# B&R Automation Studio project DuctLines (part 13)

#### Cyclic.ld
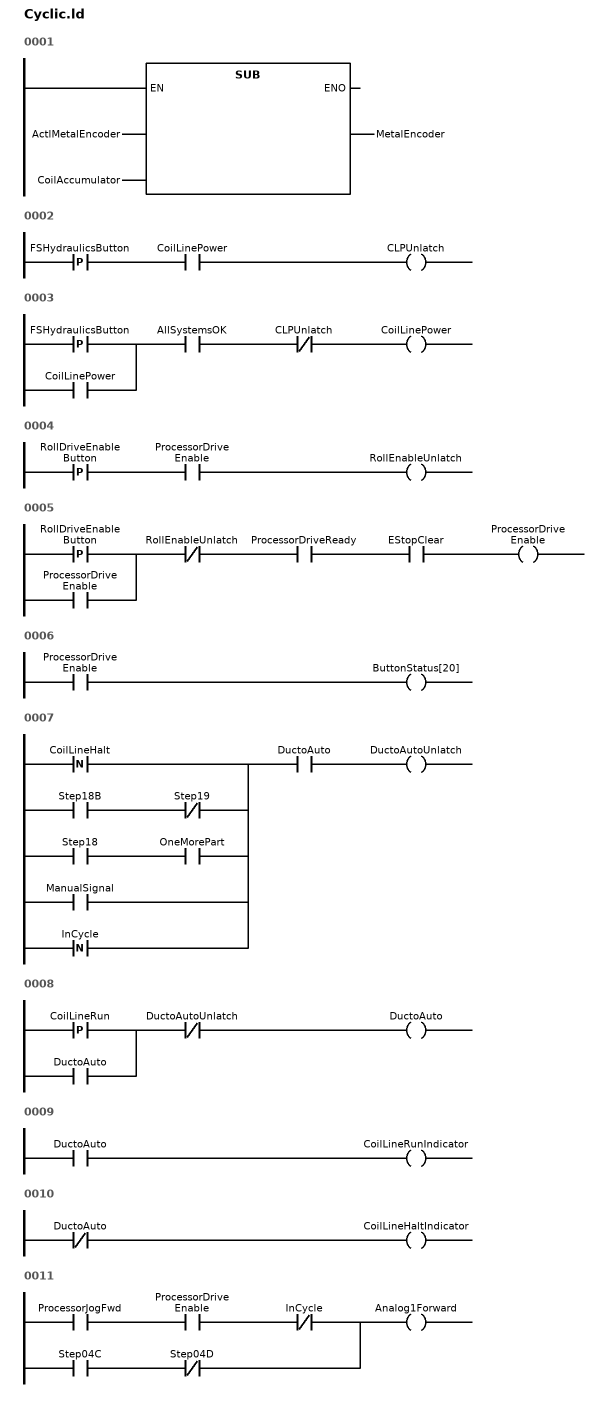
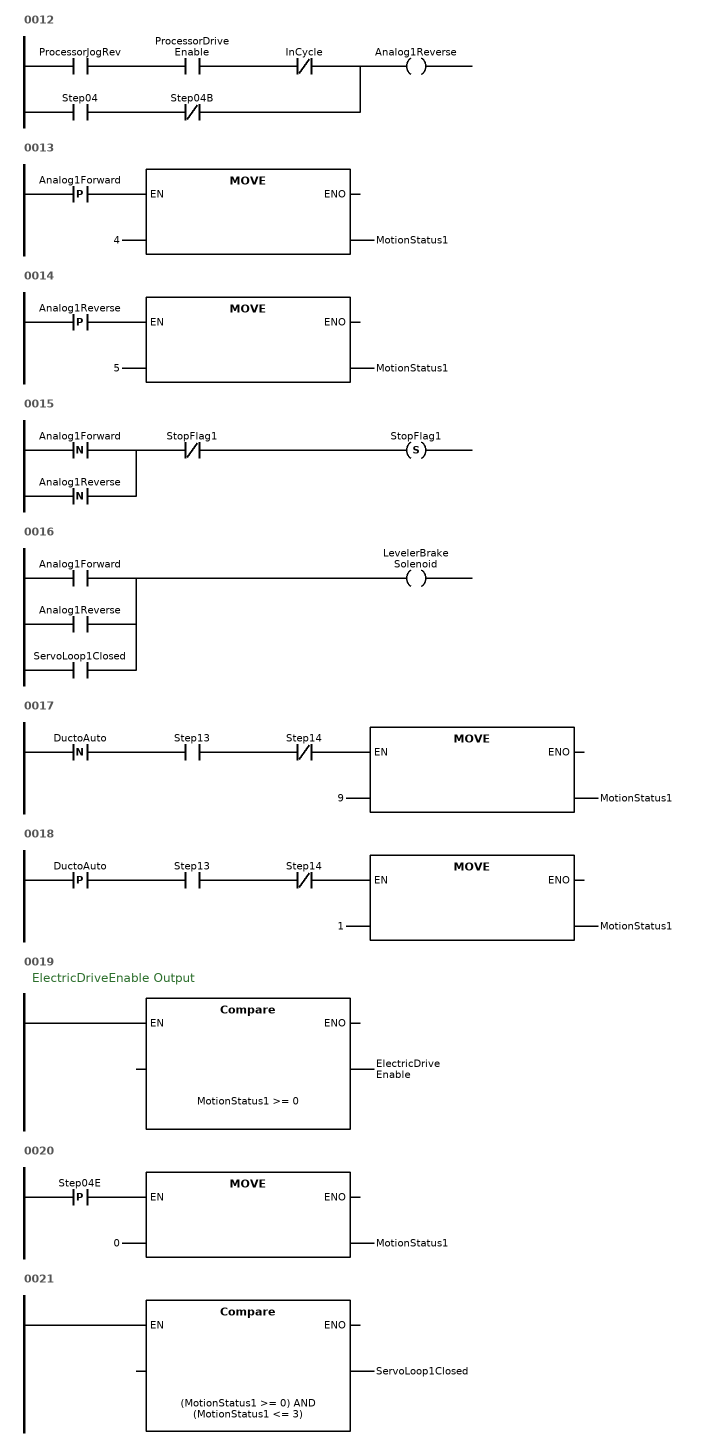
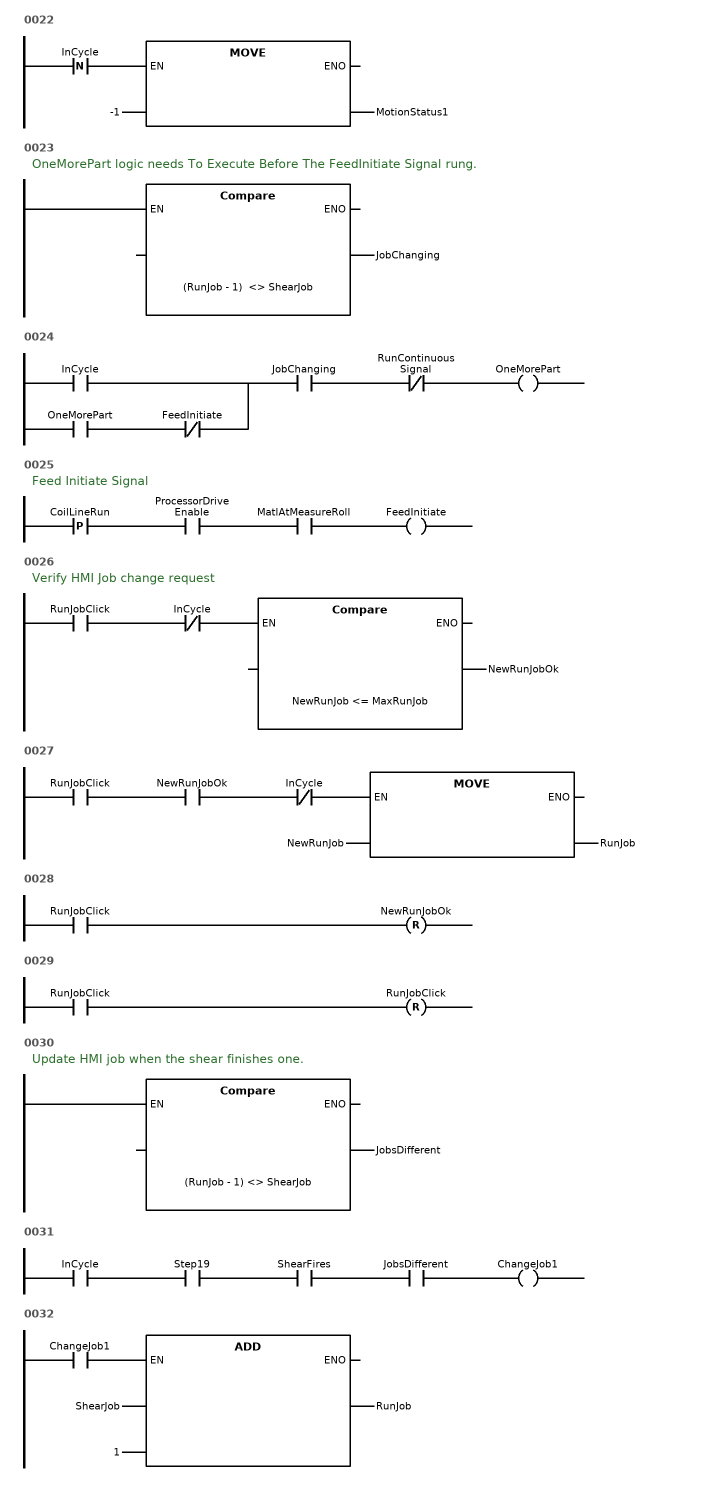
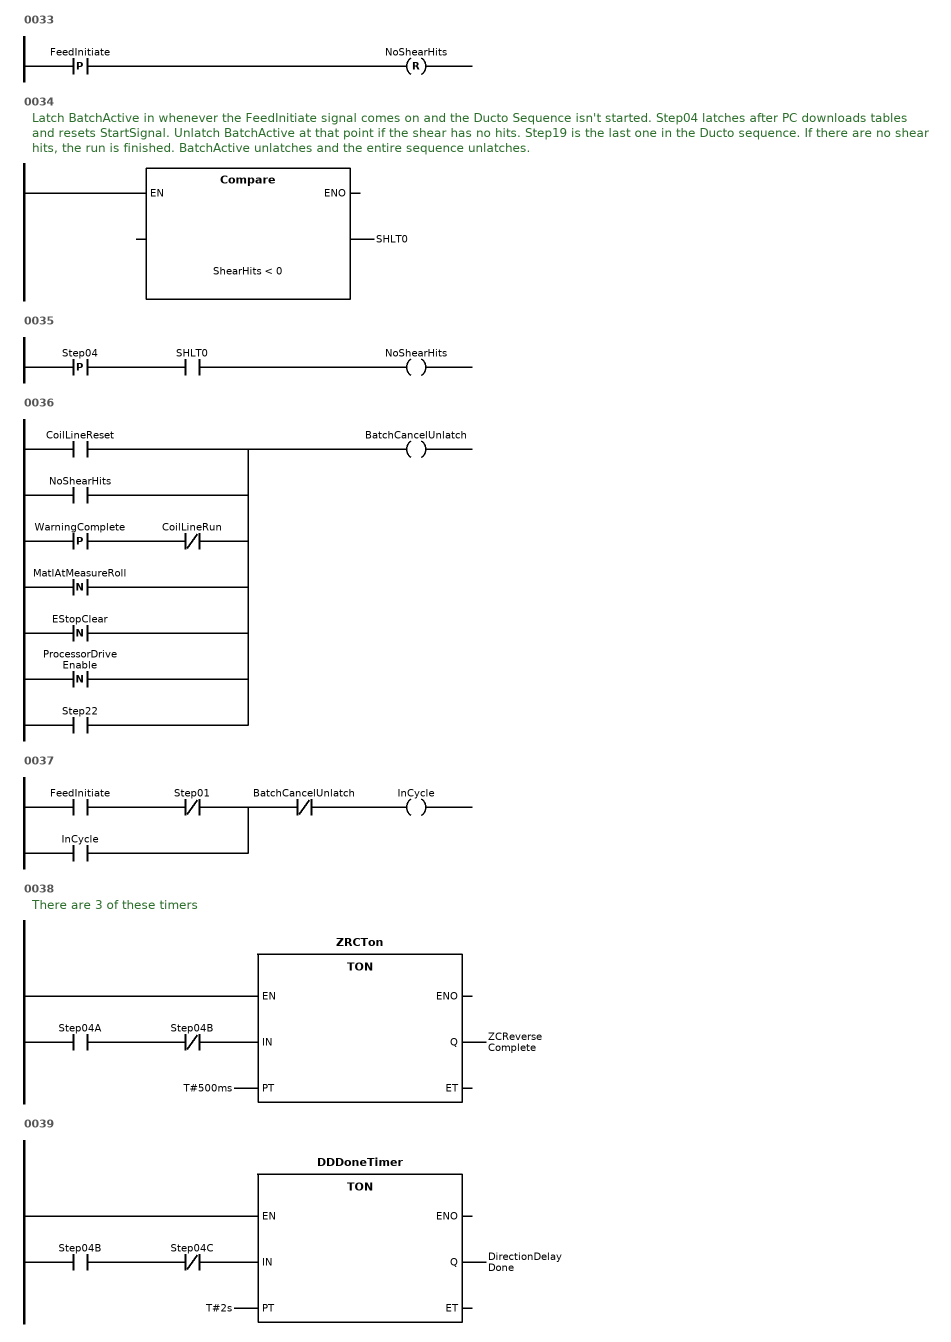
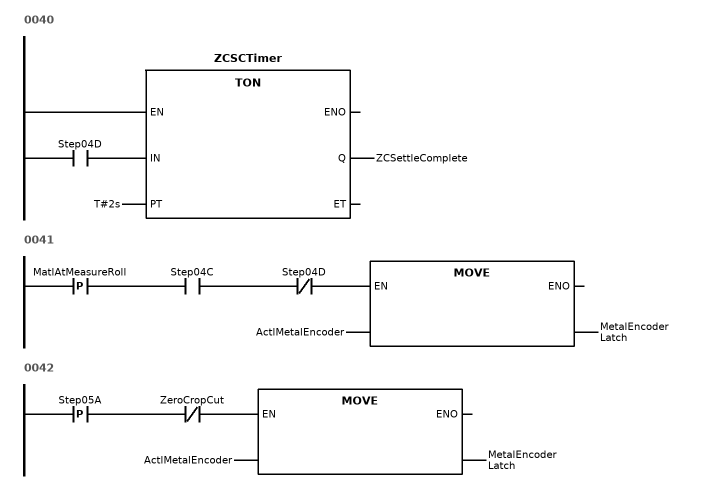
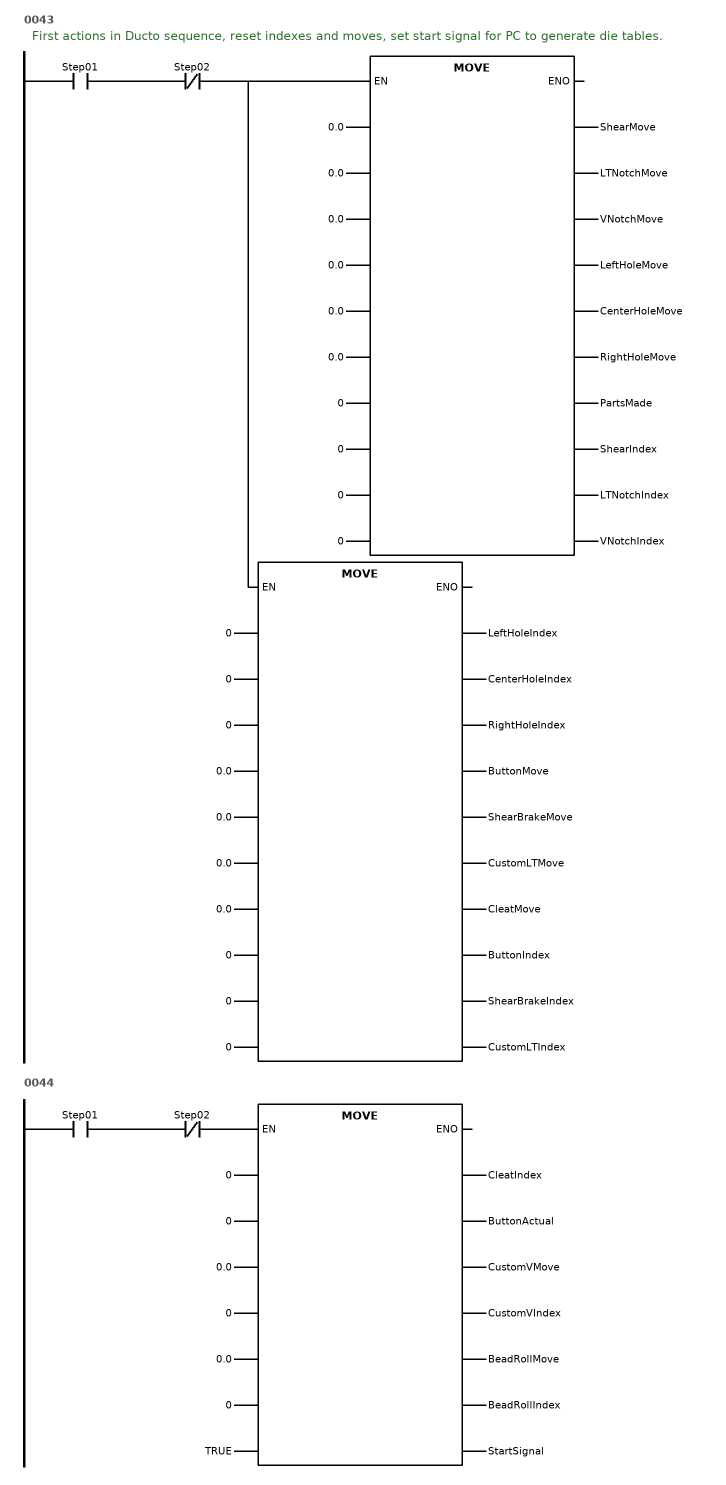
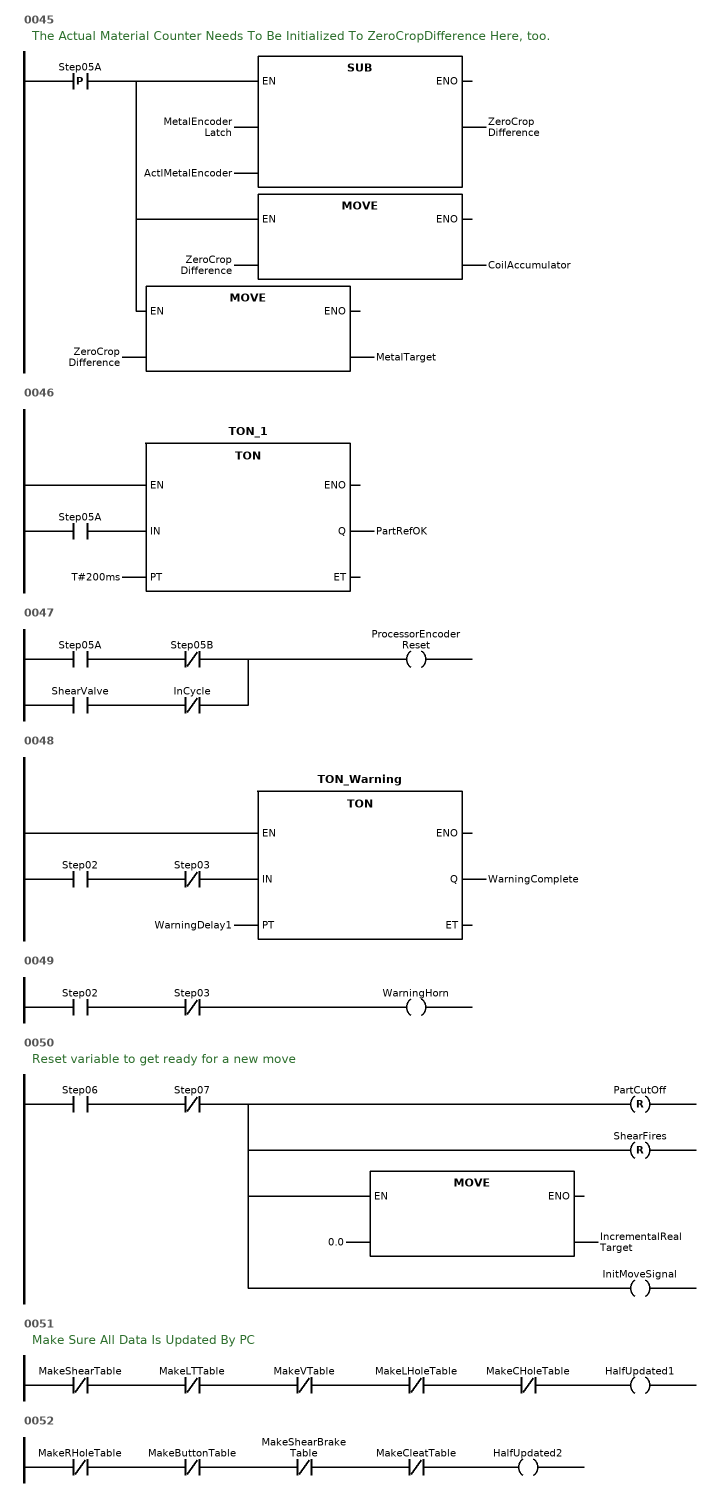
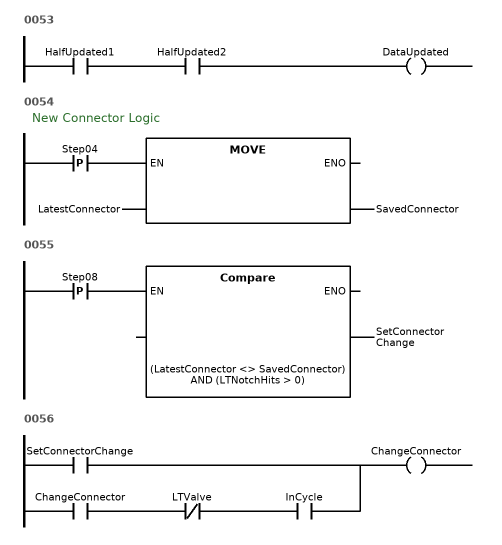
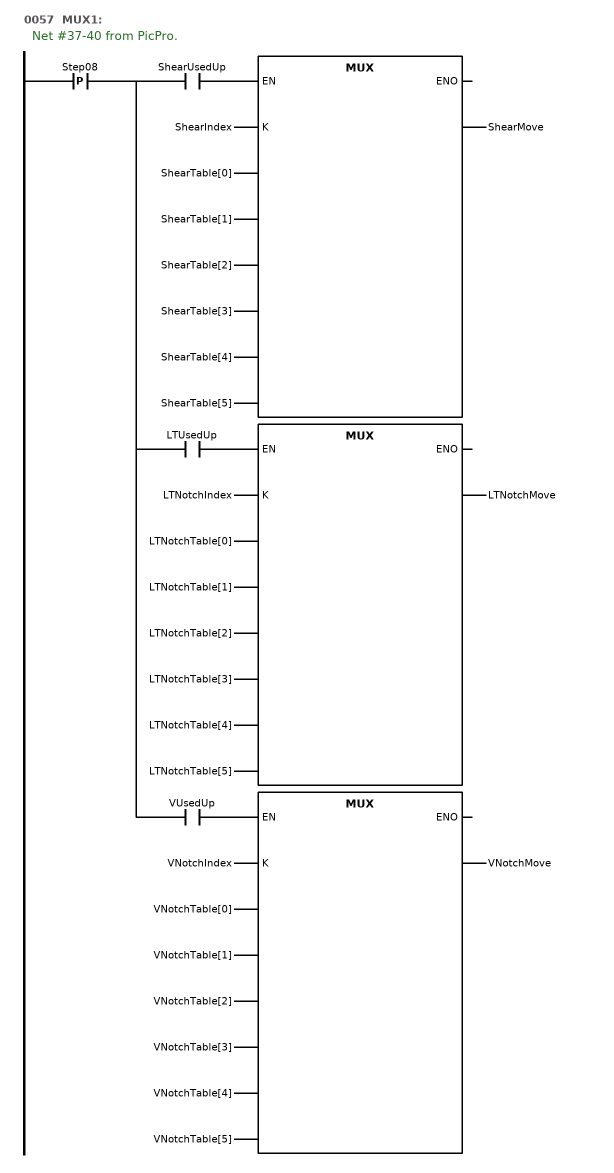
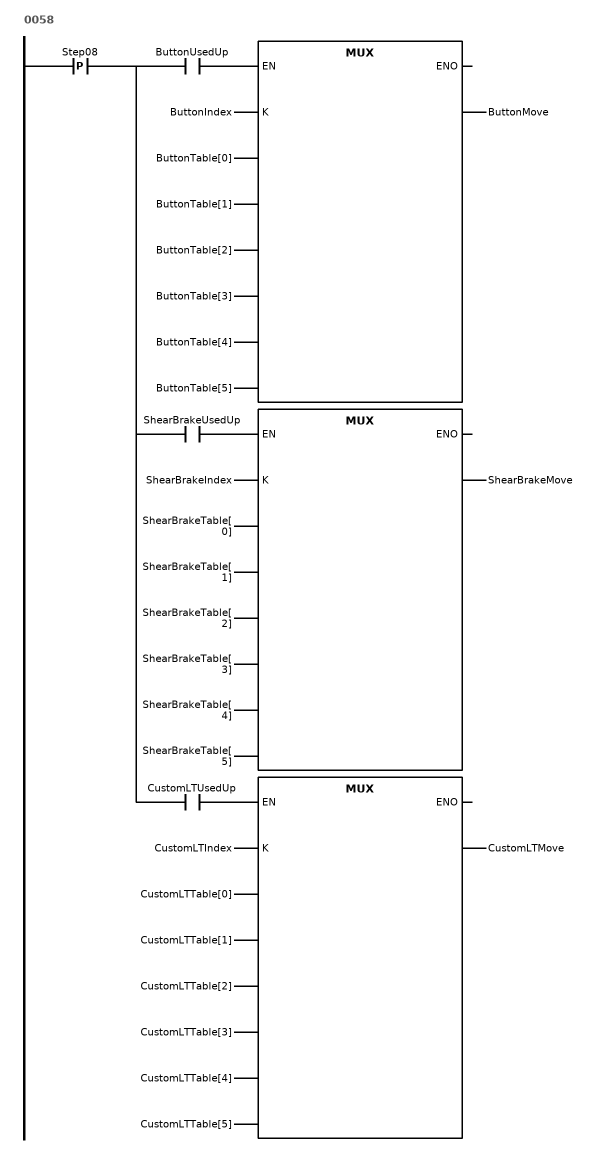
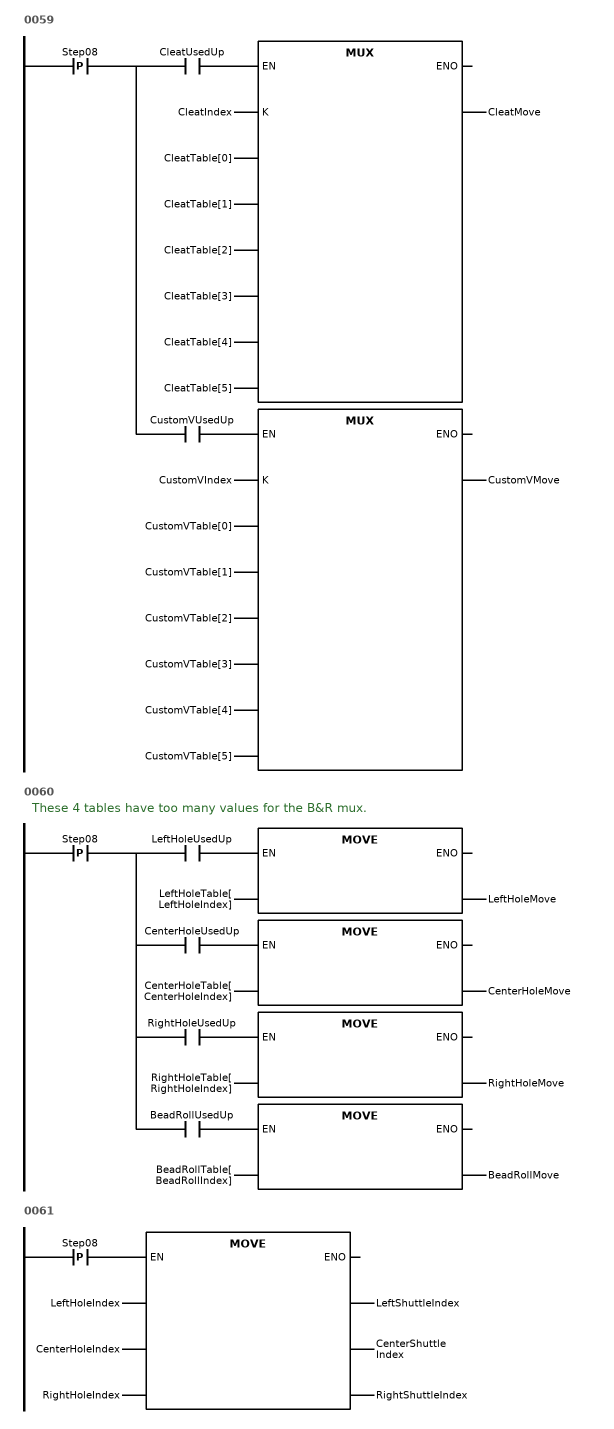
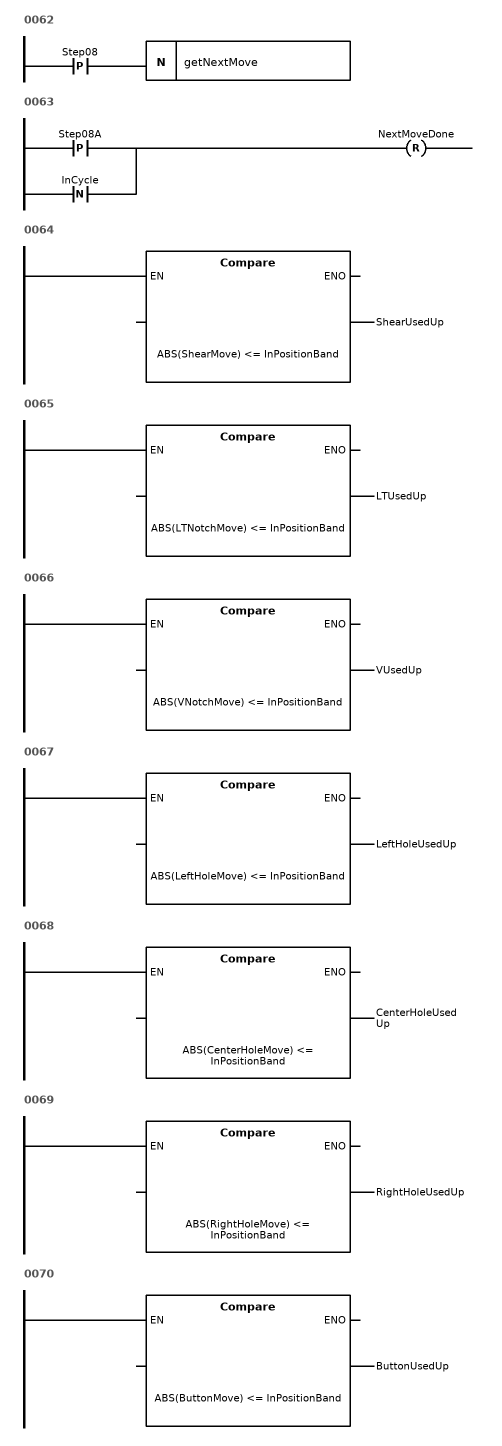
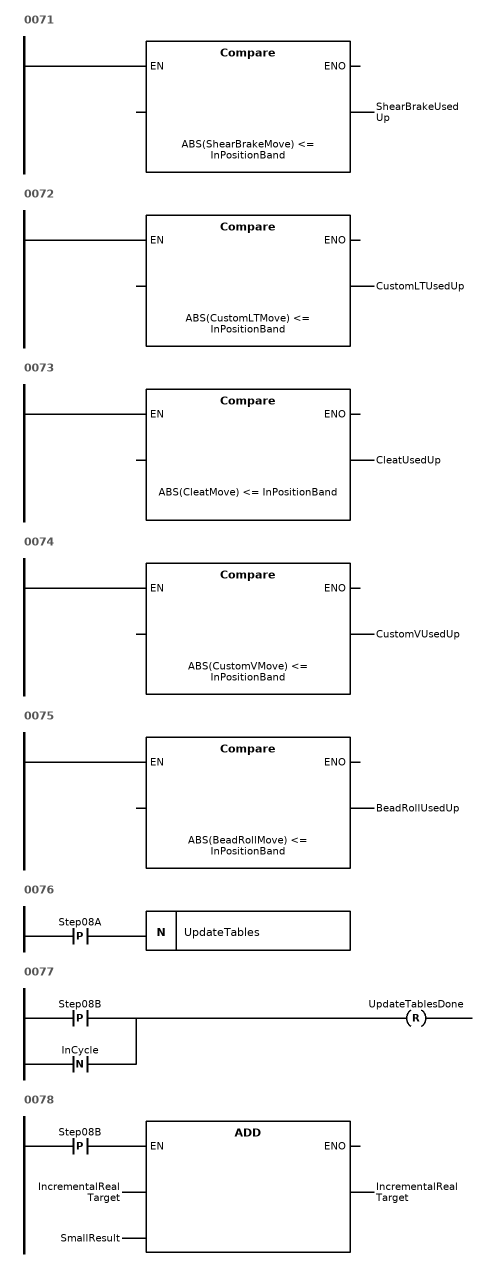
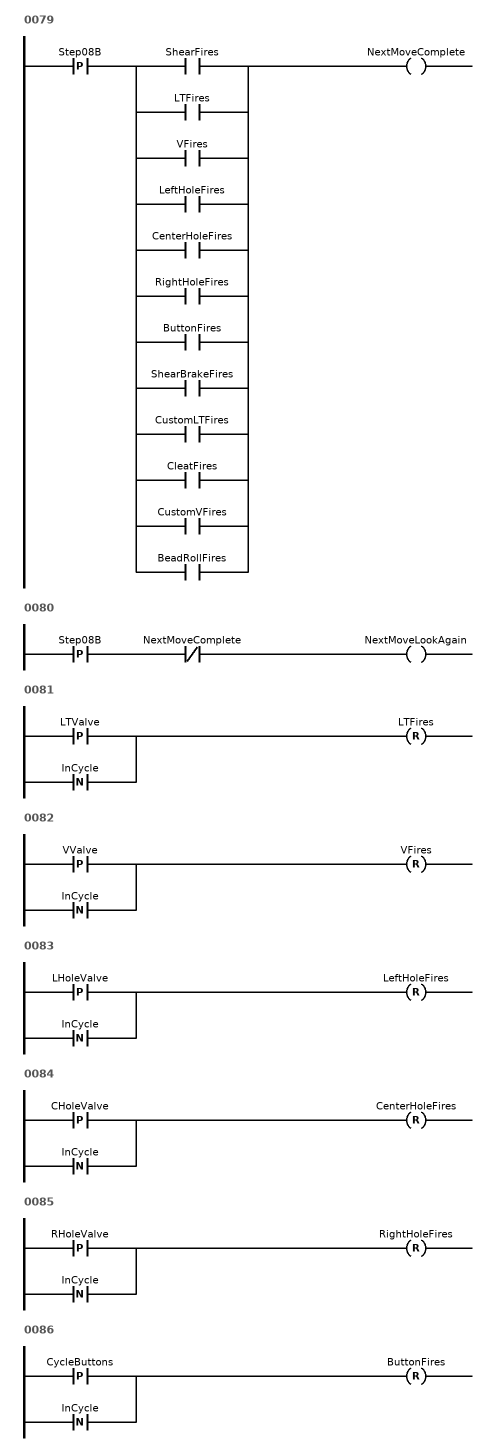
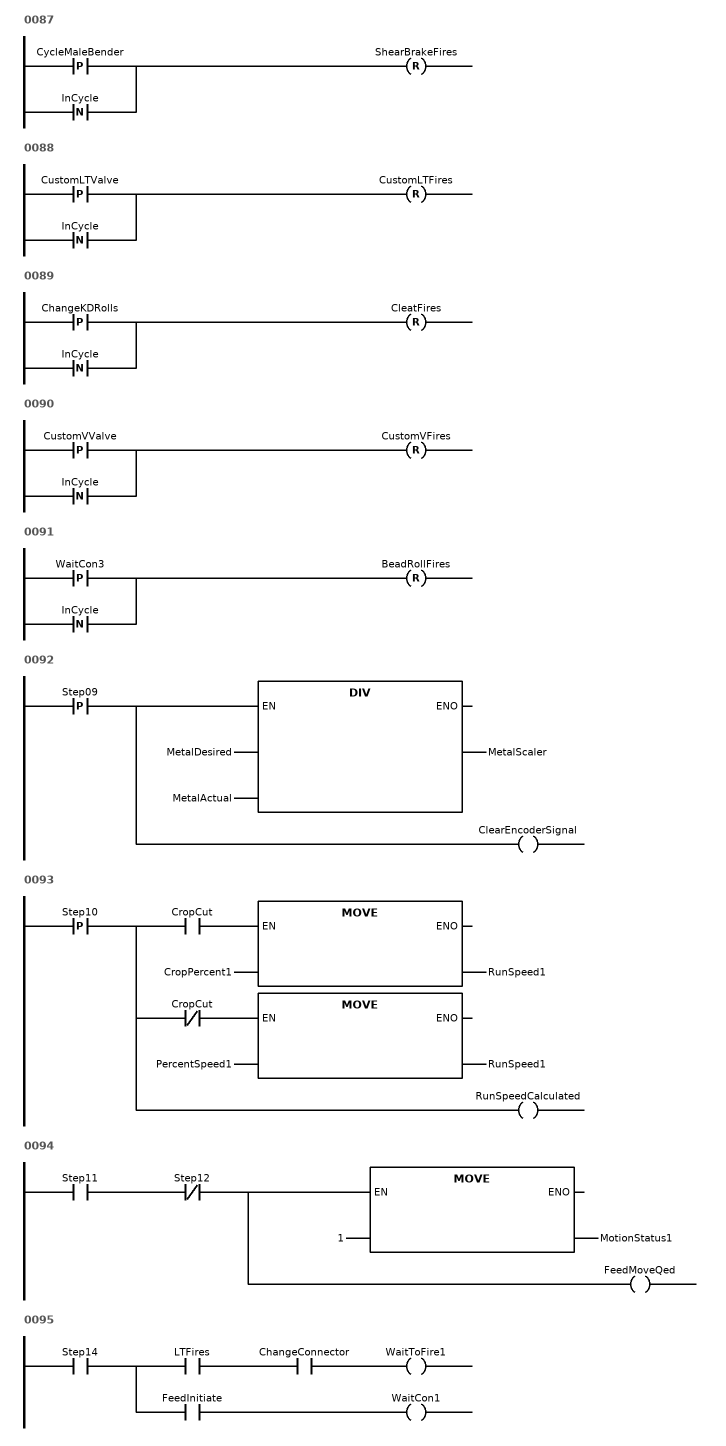
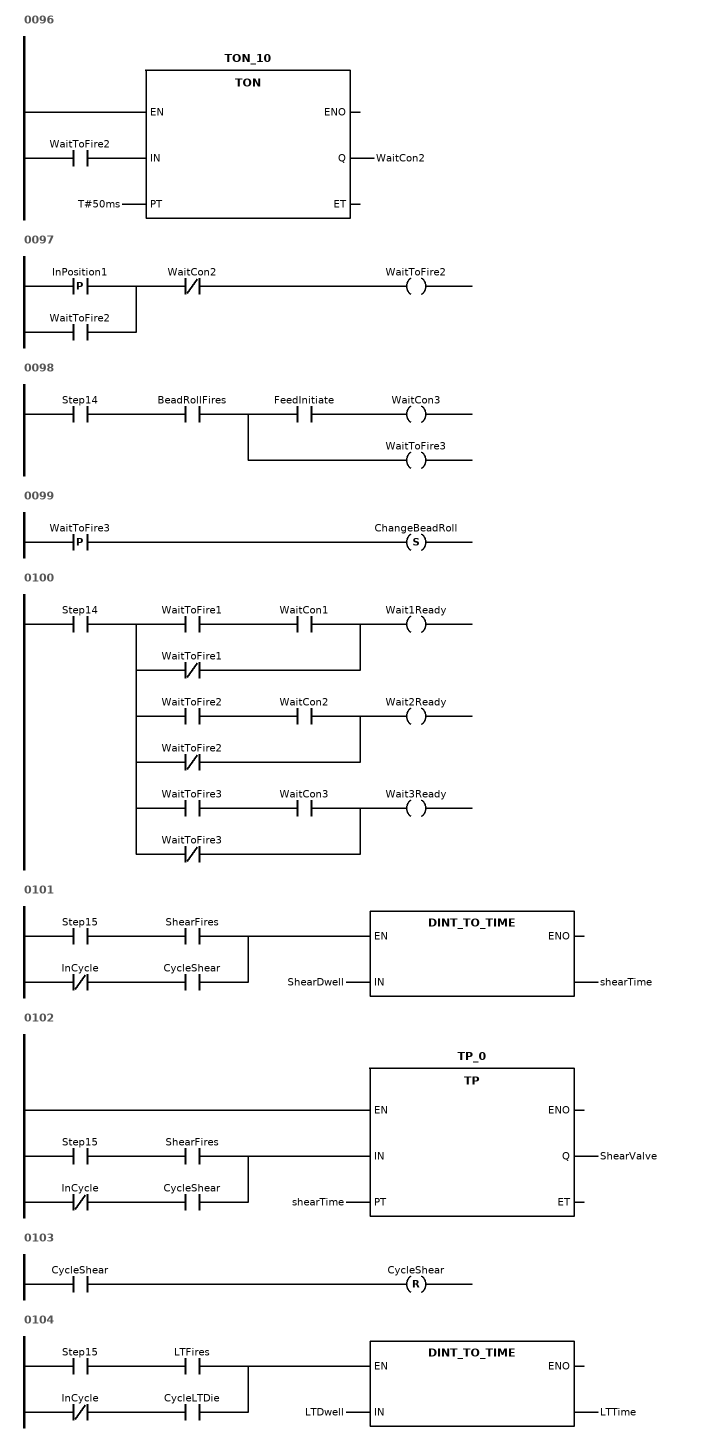
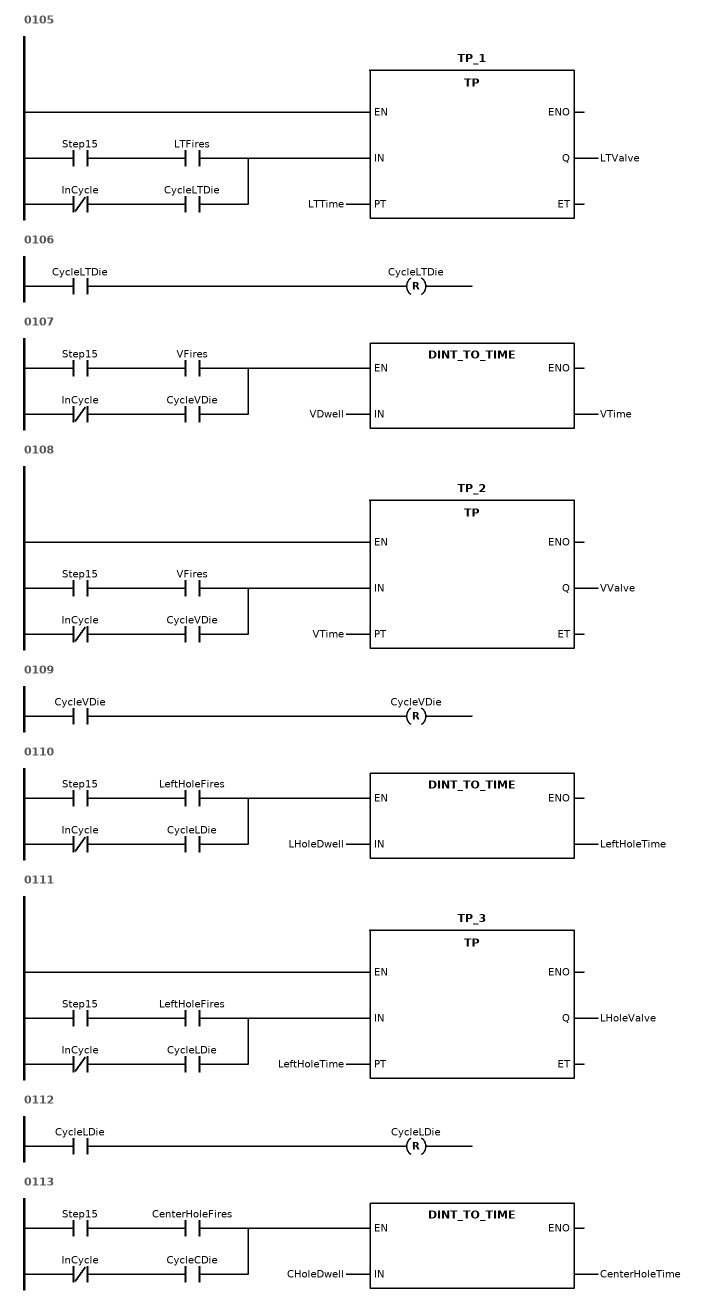
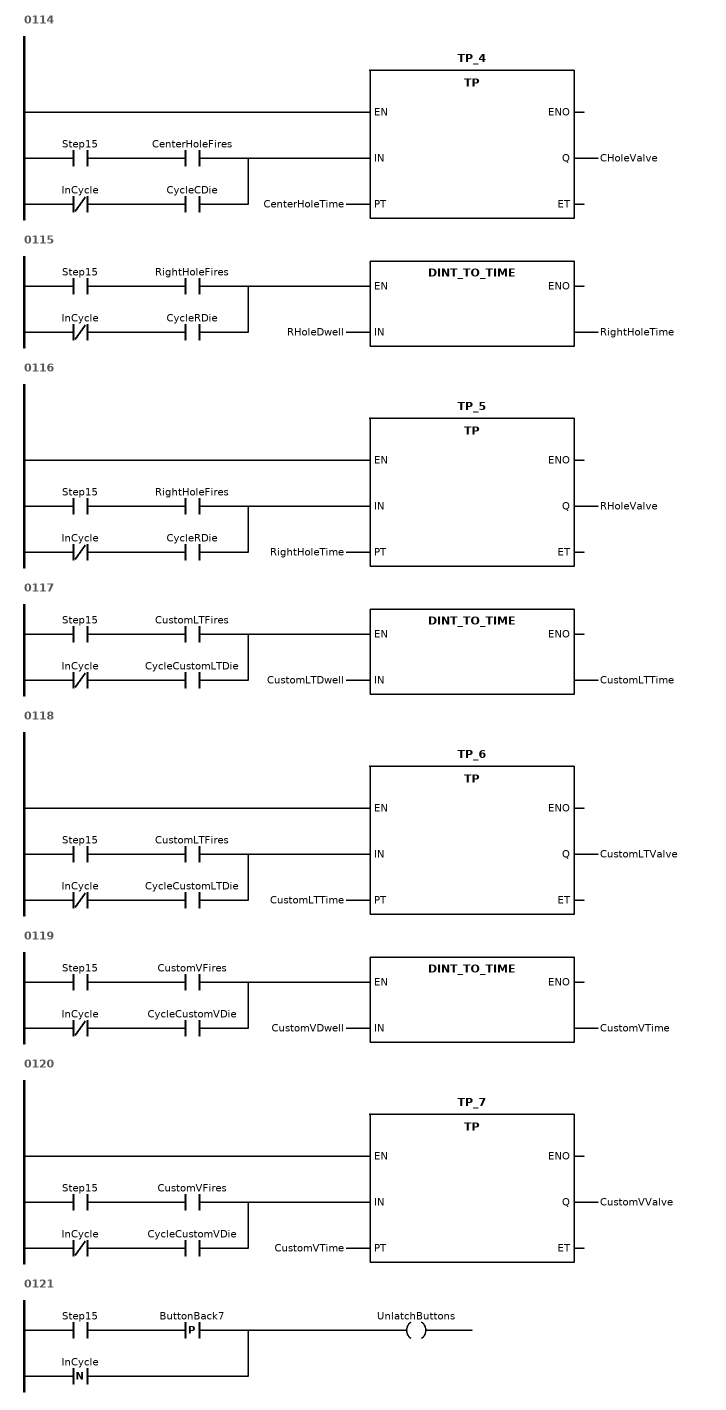
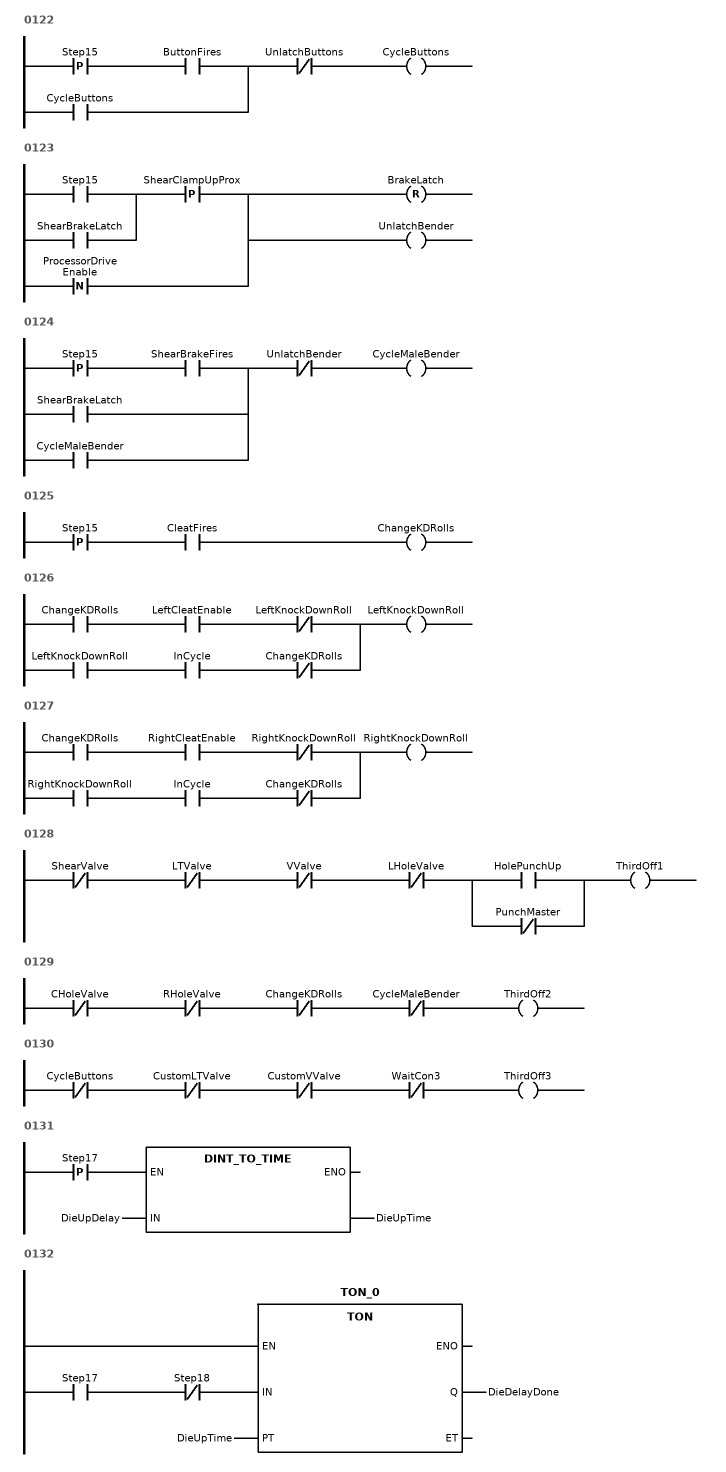
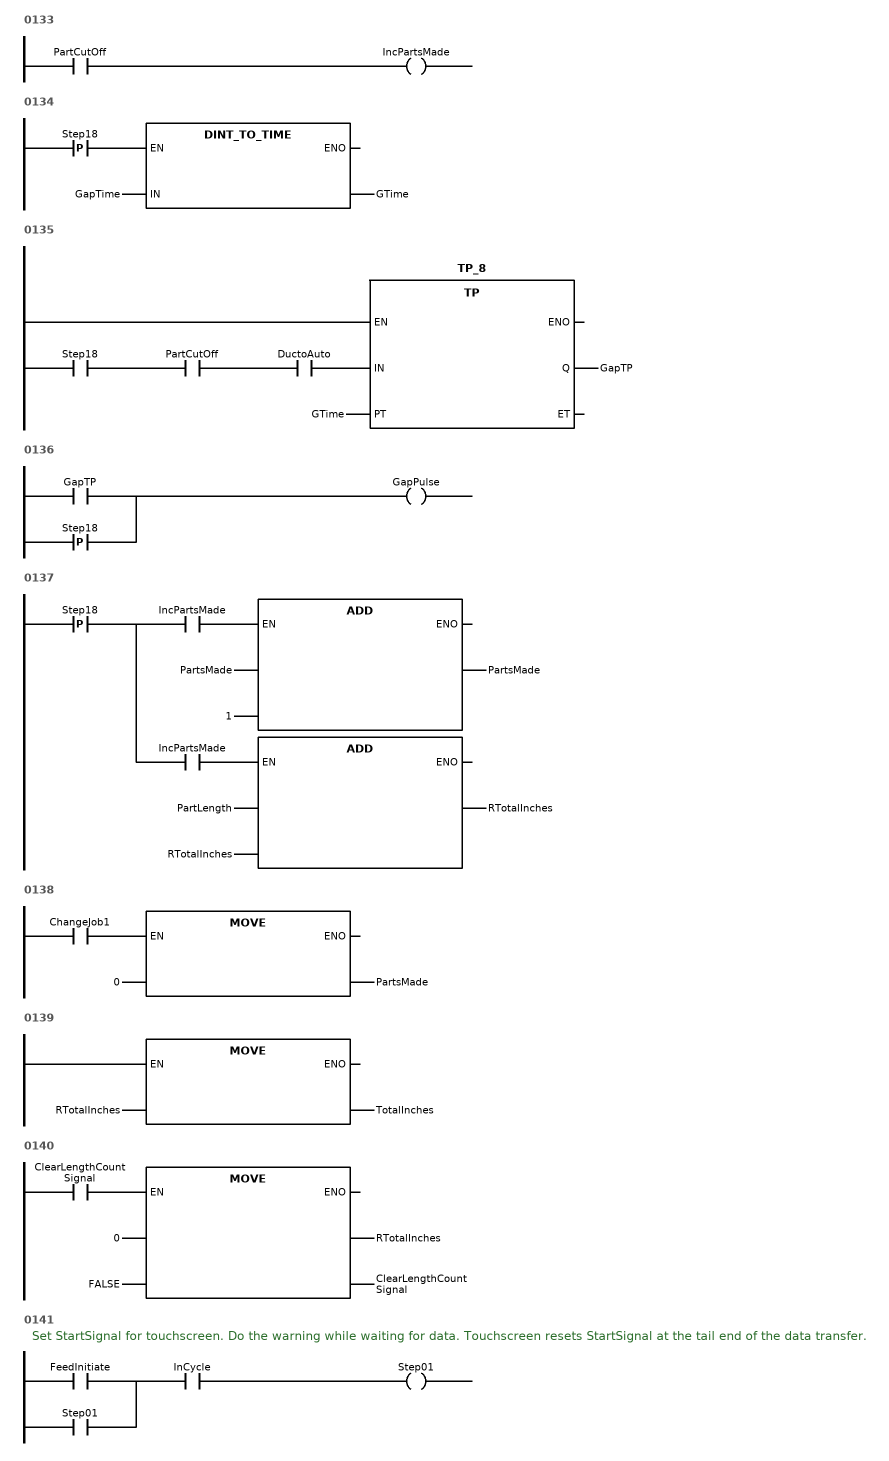
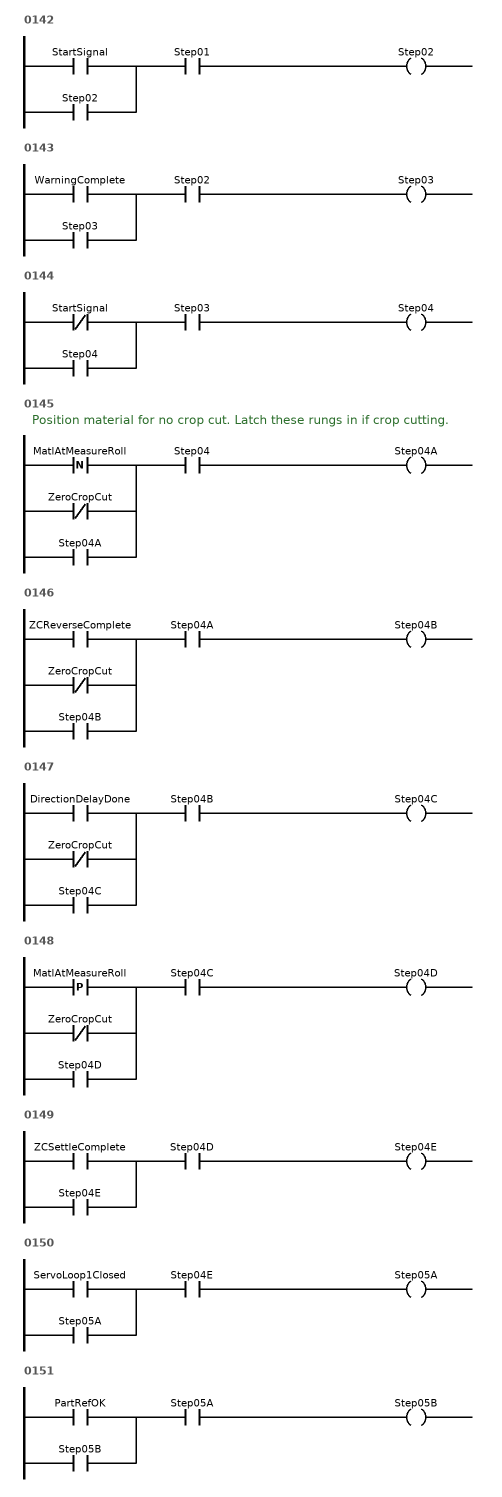
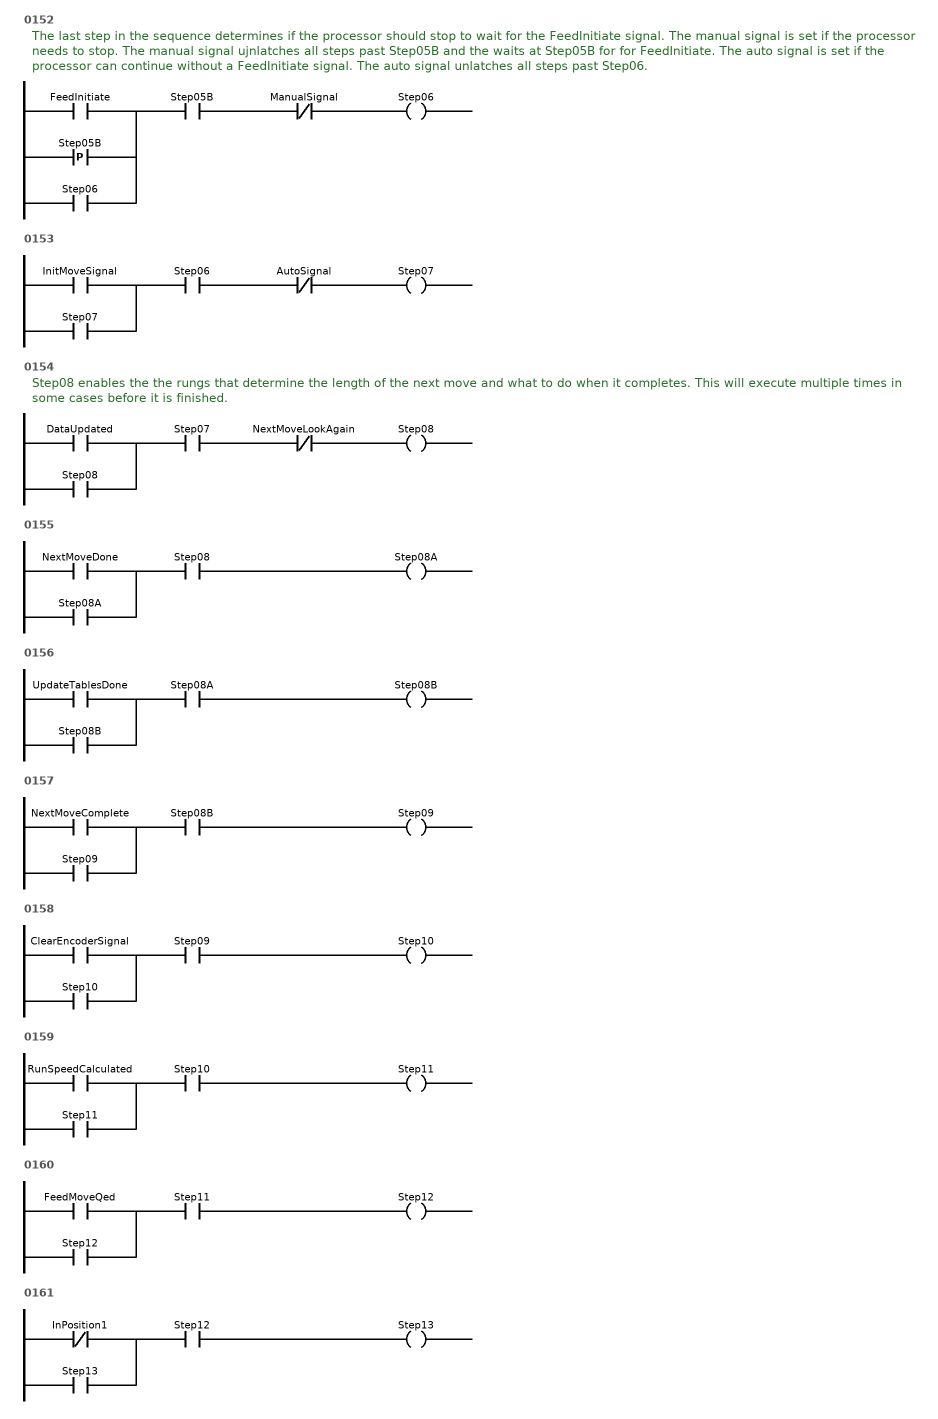
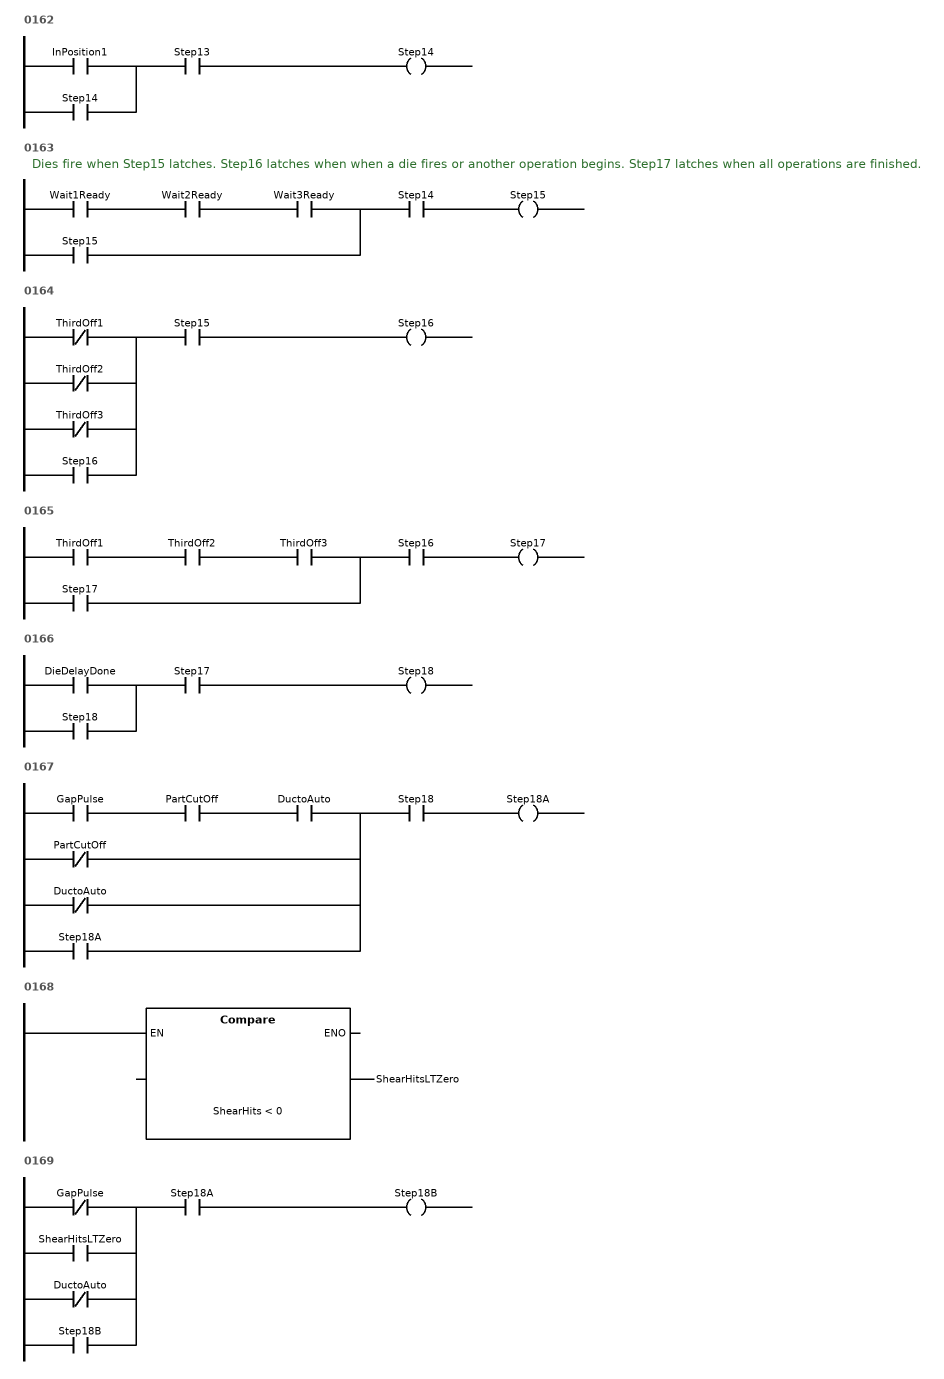
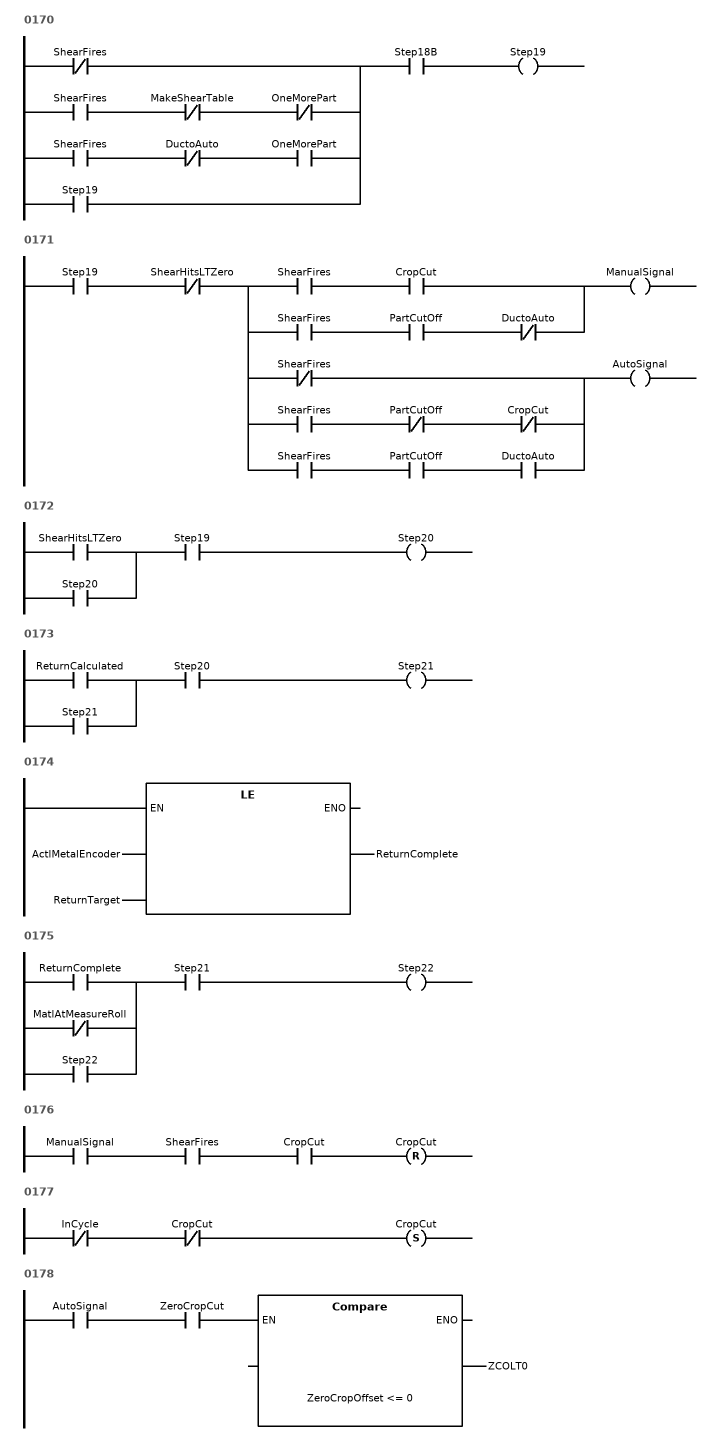
